// Mitsubishi GX Works2 project: read_high_speed   PLC: FX3U/FX3UC

PROGRAM MAIN
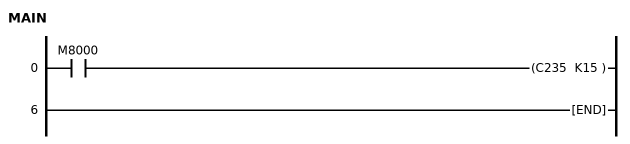
0     LD      M8000
      OUT     C235 K15
6     END
END_PROGRAM
